FUNCTION_BLOCK E_SEL_4 (* event-driven selection of data *)
  (* Standard: 61499-2; Description: An instance of an E_SEL_2 FB type provides event-driven selection of data between two inputs. Data at the OUT variable is copied from the data ( IN0 or IN1, respectively) associated with the most recent event at the EI0 or EI1 input, followed by an event at the EO output. This work is inspired by https://holobloc.com/doc/fb/rt/select/E_SEL_xxx.htm *)
  (* Version 1.0, 2024-07-03, franz *)
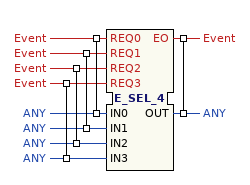
  EVENT_INPUT
    REQ0 WITH IN0;
    REQ1 WITH IN1;
    REQ2 WITH IN2;
    REQ3 WITH IN3;
  END_EVENT
  EVENT_OUTPUT
    EO WITH OUT;
  END_EVENT
  VAR_INPUT
    IN0 : ANY;
    IN1 : ANY;
    IN2 : ANY;
    IN3 : ANY;
  END_VAR
  VAR_OUTPUT
    OUT : ANY;
  END_VAR
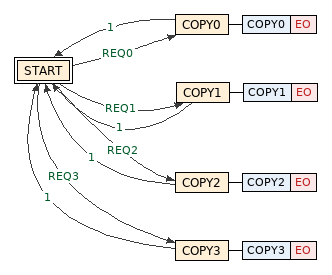
  EC_STATES
    START; (* Initial State *)
    COPY0 : COPY0 -> EO;
    COPY1 : COPY1 -> EO;
    COPY2 : COPY2 -> EO;
    COPY3 : COPY3 -> EO;
  END_STATES
  EC_TRANSITIONS
    START TO COPY0 := REQ0;
    START TO COPY1 := REQ1;
    COPY0 TO START := 1;
    COPY1 TO START := 1;
    START TO COPY2 := REQ2;
    COPY2 TO START := 1;
    START TO COPY3 := REQ3;
    COPY3 TO START := 1;
  END_TRANSITIONS
  ALGORITHM COPY0 IN ST:
OUT := IN0;
  END_ALGORITHM
  ALGORITHM COPY1 IN ST:
OUT := IN1;
  END_ALGORITHM
  ALGORITHM COPY2 IN ST:
OUT := IN2;
  END_ALGORITHM
  ALGORITHM COPY3 IN ST:
OUT := IN3;
  END_ALGORITHM
END_FUNCTION_BLOCK
